{attribute 'linkalways'} 
{attribute 'no_explicit_call' := 'This FB is a CLASS and must be accessed using methods or properties'}
{attribute 'enable_dynamic_creation'}
FUNCTION_BLOCK _ETcVnEstimationAlgorithm EXTENDS EnumDatatypeBase
VAR
	localData : ETcVnEstimationAlgorithm;
	activeData : REFERENCE TO ETcVnEstimationAlgorithm;
	enumBaseDatatype : _DINT(localData);
END_VAR

METHOD PRIVATE AddLocalEnumeration
VAR_INPUT
	Enumeration : T_MAXSTRING;
	Value : ETcVnEstimationAlgorithm;
END_VAR
AddEnumeration(Enumeration, Value);
END_METHOD

PROPERTY PUBLIC Address : PVOID
GET
Address := ADR(activeData);
END_GET
END_PROPERTY

METHOD PUBLIC ClearReference
VAR_INPUT
END_VAR
activeData REF= localData;
SetBaseDatatypeReference();
END_METHOD

METHOD PUBLIC Clone : I_Datatype
VAR
    pClone : POINTER TO _ETcVnEstimationAlgorithm;
END_VAR
pClone := __NEW(_ETcVnEstimationAlgorithm(InitialValue := Value));
Clone := pClone^;
END_METHOD

METHOD FB_init : BOOL
VAR_INPUT
	bInitRetains : BOOL; // if TRUE, the retain variables are initialized (warm start / cold start)
	bInCopyCode : BOOL;  // if TRUE, the instance afterwards gets moved into the copy code (online change)
	InitialValue : ETcVnEstimationAlgorithm;
END_VAR
localData := InitialValue;
AddBaseDatatype(enumBaseDatatype);
ClearReference();

AddLocalEnumeration('TCVN_EA_DEFAULT', ETcVnEstimationAlgorithm.TCVN_EA_DEFAULT);
AddLocalEnumeration('TCVN_EA_LMEDS', ETcVnEstimationAlgorithm.TCVN_EA_LMEDS);
AddLocalEnumeration('TCVN_EA_RANSAC', ETcVnEstimationAlgorithm.TCVN_EA_RANSAC);
AddLocalEnumeration('TCVN_EA_RHO', ETcVnEstimationAlgorithm.TCVN_EA_RHO);
END_METHOD

PROPERTY PUBLIC Identifier : T_MAXSTRING
GET
Identifier := 'ETcVnEstimationAlgorithm';
END_GET
END_PROPERTY

METHOD IsEnumeratorValueEqual : BOOL
VAR_INPUT
	Enumerator : I_KeyValueForwardEnumerator;
END_VAR
VAR
	storedValue : ETcVnEstimationAlgorithm;
END_VAR
IF NOT Enumerator.TryGet(storedValue) THEN
	RETURN;
END_IF

IsEnumeratorValueEqual := storedValue = activeData;
END_METHOD

METHOD PUBLIC MakeReferenceTo
VAR_INPUT
	ReferenceTarget : REFERENCE TO ETcVnEstimationAlgorithm;
END_VAR
activeData REF= ReferenceTarget;
SetBaseDatatypeReference();
END_METHOD

METHOD PROTECTED SetBaseDatatypeReference
VAR_INPUT
END_VAR
enumBaseDatatype.MakeReferenceTo(activeData);
END_METHOD

PROPERTY PUBLIC Size : UDINT
GET
Size := SIZEOF(activeData);
END_GET
END_PROPERTY

METHOD TryMakeReferenceTo : BOOL
VAR_INPUT
	Target : I_Datatype;
END_VAR
VAR
	pTargetData : POINTER TO ETcVnEstimationAlgorithm;
END_VAR
IF NOT IsEquivalentTo(Target) THEN
	RETURN;
END_IF

pTargetData := Target.Address;
activeData REF= pTargetData^;
SetBaseDatatypeReference();
TryMakeReferenceTo := TRUE;
END_METHOD

PROPERTY PUBLIC Value : ETcVnEstimationAlgorithm
GET
Value := activeData;
END_GET
SET
activeData := Value;
END_SET
END_PROPERTY

END_FUNCTION_BLOCK

(* stored: Version 1.1.0.1, ProductVersion 3.1.4024.13
   POU _ETcVnEstimationAlgorithm: Id {7f908390-7cf4-0c40-3e4e-88fc3549b526}, SpecialFunc None
   Folder Core: Id {26e06ea9-f338-0d7f-0553-ab085d985d08}
   Folder Protected: Id {751d3d80-21d3-0083-2916-f8ee13d1e9fa}
   Folder Customize: Id {ad2e4fac-c5b0-036b-0a7a-fa78cc16a697}
   Folder Constructor: Id {f3bdf0bc-ef44-0f68-3edc-e6c7c40f8b82}
   Folder Private: Id {36981ce6-6862-0a68-1a52-03c1caa00aa8}
   Folder Protected: Id {a9069b81-c089-09c7-2c68-af8da621324c}
   Method AddLocalEnumeration: Id {1e40741b-3d87-0f9f-30cd-674a66451e32}
   Property Address: Id {a354e235-384b-0e24-2348-7053e28704cc}
   Get Get: Id {725164f9-cd22-0be7-2eb5-22280b27fe1a}
   Method ClearReference: Id {733b4b09-5d82-0a5c-0295-11d7aa39bc54}
   Method Clone: Id {c2a76f91-e717-0982-2f22-940600b513d6}
   Method FB_init: Id {01701bed-115a-01b0-11dd-15c61e5d3ff5}
   Property Identifier: Id {c71245ca-ca0d-07b4-2a38-3b4d3467fccc}
   Get Get: Id {d6257192-c389-0847-3b39-861e7d0a4848}
   Method IsEnumeratorValueEqual: Id {7b472005-ed96-0203-1764-19759411abfd}
   Method MakeReferenceTo: Id {af0b78d7-1ed7-0b79-2279-457a6cbcf851}
   Method SetBaseDatatypeReference: Id {5e785bc7-f839-025c-1fde-5874d9366a0b}
   Property Size: Id {7413c091-3481-095e-3b89-29e8452d2394}
   Get Get: Id {819b0509-7065-06b4-25cb-fafb0524b639}
   Method TryMakeReferenceTo: Id {0ba35ee4-2308-061c-38d8-6d47caa923c0}
   Property Value: Id {59aae314-2ccd-0a2f-3d57-7e0140d2ae76}
   Get Get: Id {35aedeee-f2b6-09a9-2e4b-b5f403a04edc}
   Set Set: Id {900a5a3d-4468-056f-22c4-ccfed841dcd3} *)
